(* PLC project Generated.project, CODESYS CODESYS V3.5 SP19 Patch 1 *)
(* stored: creationDateTime 2026-09-06T13:00:42.431888, modificationDateTime 2026-09-06T13:00:42.431888 *)

(* ======================================================================= ⚖️ ST_fbWinch_Symmetry_Cfg — Configuration des seuils de symétrie M1/M2 ─────────────────────────────────────────────────────────────── 🎯 Rôle : Seuils de tolérance pour le diagnostic passif de symétrie treuils 📄 Doc métier : DOC/AF/AF_Partie-10_Fonction_Winch_v2.1.md ======================================================================= *)
TYPE ST_fbWinch_Symmetry_Cfg : STRUCT
  DeltaStartDelay_Ms : UDINT := 100;  (* Ecart max tolere au demarrage (ms) *)
  DeltaBrakeReleaseTime_Ms : UDINT := 100;  (* Ecart max temps desserrage frein (ms) *)
  DeltaBrakeApplyTime_Ms : UDINT := 100;  (* Ecart max temps serrage frein (ms) *)
  DeltaStopDistance_Mm : UDINT := 100;  (* Ecart max distance d'arret (mm) *)
  DeltaStopTime_Ms : UDINT := 200;  (* Ecart max temps d'arret (ms) *)
  MinimumCommandTime_Ms : UDINT := 1000;  (* Duree minimale de commande pour qualification (ms) *)
  MinimumSpeed_Mps : REAL := 0.05;  (* Vitesse minimale pour qualification (m/s) *)
END_STRUCT;
END_TYPE

(* ======================================================================= 📊 ST_fbWinch_Symmetry_Data — Données mesurées de symétrie M1/M2 ─────────────────────────────────────────────────────────────── 🎯 Rôle : Structure des résultats de mesures et d'écarts du diagnostic symétrie 📄 Doc métier : DOC/AF/AF_Partie-10_Fonction_Winch_v2.1.md ======================================================================= *)
TYPE ST_fbWinch_Symmetry_Data : STRUCT
  DeltaStartDelay_Ms : UDINT;  (* Ecart mesure au demarrage (ms) *)
  DeltaBrakeReleaseTime_Ms : UDINT;  (* Ecart mesure temps desserrage frein (ms) *)
  DeltaBrakeApplyTime_Ms : UDINT;  (* Ecart mesure temps serrage frein (ms) *)
  DeltaStopDistance_Mm : UDINT;  (* Ecart mesure distance d'arret (mm) *)
  DeltaStopTime_Ms : UDINT;  (* Ecart mesure temps d'arret (ms) *)
  MaxSyncDeviation_M : REAL;  (* Ecart maximal de synchronisme enregistre (m) *)
END_STRUCT;
END_TYPE

(* ======================================================================= ⚖️ FB_Winch_Symmetry — Mesure passive M1/M2 ─────────────────────────────────────────────────────────────── 🎯 Rôle : Observateur de symétrie et de synchronisme des treuils M1/M2 📄 Doc métier : DOC/AF/AF_Partie-10_Fonction_Winch_v2.1.md 🔒 Observateur pur : Aucune ecriture de commande, securite ou mouvement ======================================================================= *)
FUNCTION_BLOCK FB_Winch_Symmetry
  VAR_INPUT
    Reset : BOOL;  (* === COMMANDES ET CONSIGNES === --> [CMD] Reinitialisation des mesures sur front *)
    M1CommandActive : BOOL;  (* --> [CMD] Commande active sur treuil M1 *)
    M2CommandActive : BOOL;  (* --> [CMD] Commande active sur treuil M2 *)
    M1Direction : INT;  (* --> [CMD] Sens commande M1 (-1/0/+1) *)
    M2Direction : INT;  (* --> [CMD] Sens commande M2 (-1/0/+1) *)
    M1BrakeCmd : BOOL;  (* === FEEDBACKS HARWARE ET FREINS === --> [HW] Ordre ouverture frein M1 *)
    M2BrakeCmd : BOOL;  (* --> [HW] Ordre ouverture frein M2 *)
    M1BrakeApplied : BOOL;  (* --> [HW] Etat frein M1 serre *)
    M2BrakeApplied : BOOL;  (* --> [HW] Etat frein M2 serre *)
    M1Position_M : REAL;  (* === MESURES POSITIONS ET VITESSES === --> [HW] Position mesuree M1 (m) *)
    M2Position_M : REAL;  (* --> [HW] Position mesuree M2 (m) *)
    M1Speed_Mps : REAL;  (* --> [HW] Vitesse mesuree M1 (m/s) *)
    M2Speed_Mps : REAL;  (* --> [HW] Vitesse mesuree M2 (m/s) *)
    SyncDeviation_M : REAL;  (* --> [HW] Ecart instantane synchro (m) *)
    Config : ST_fbWinch_Symmetry_Cfg;  (* === CONFIGURATION === --> [CFG] Configuration des seuils de symetrie *)
  END_VAR
  VAR_OUTPUT
    SymmetryOk : BOOL;  (* === ETATS IEC ET SYNOPTIQUE === <-- [STAT] Symetrie globale conforme aux criteres *)
    SymmetryValid : BOOL;  (* <-- [STAT] Mesure de symetrie valide et calculee *)
  END_VAR
  VAR_IN_OUT
    Data : ST_fbWinch_Symmetry_Data;  (* === STRUCTURES DE DONNÉES PARTAGÉES === <-> [BUS] Donnees de mesures de symetrie *)
  END_VAR
  VAR
    ResetEdge : R_TRIG;  (* === SOUS-INSTANCES FB === * [INST] Detecteur front reinitialisation *)
    CycleTime : FB_CycleTime;  (* * [INST] Calcul du temps de cycle *)
    CommandTon : TON;  (* === TIMERS INTERNES === . [LOC] Tempo qualification commande stable *)
    MotionTimer : TON;  (* . [LOC] Chronometre de mouvement *)
    StopTimer : TON;  (* . [LOC] Chronometre d'arret *)
    Comparable : BOOL;  (* === VARIABLES LOCALES CALCULÉES === . [LOC] Conditions de comparaison remplies *)
    Qualified : BOOL;  (* . [LOC] Phase de mesure qualifiee *)
    PreviousQualified : BOOL;  (* . [LOC] Etat qualifie cycle precedent *)
    Stopping : BOOL;  (* . [LOC] Phase d'arret en cours *)
    StartCapturedM1 : BOOL;  (* . [LOC] Top depart capture M1 *)
    StartCapturedM2 : BOOL;  (* . [LOC] Top depart capture M2 *)
    StopCapturedM1 : BOOL;  (* . [LOC] Top arret capture M1 *)
    StopCapturedM2 : BOOL;  (* . [LOC] Top arret capture M2 *)
    StartMsM1 : UDINT;  (* . [LOC] Horodatage d'ouverture M1 (ms) *)
    StartMsM2 : UDINT;  (* . [LOC] Horodatage d'ouverture M2 (ms) *)
    ReleaseMsM1 : UDINT;  (* . [LOC] Temps de desserrage frein M1 (ms) *)
    ReleaseMsM2 : UDINT;  (* . [LOC] Temps de desserrage frein M2 (ms) *)
    ApplyMsM1 : UDINT;  (* . [LOC] Temps de serrage frein M1 (ms) *)
    ApplyMsM2 : UDINT;  (* . [LOC] Temps de serrage frein M2 (ms) *)
    StopMsM1 : UDINT;  (* . [LOC] Horodatage d'arret M1 (ms) *)
    StopMsM2 : UDINT;  (* . [LOC] Horodatage d'arret M2 (ms) *)
    StopStartM1_M : REAL;  (* . [LOC] Position debut d'arret M1 (m) *)
    StopStartM2_M : REAL;  (* . [LOC] Position debut d'arret M2 (m) *)
  END_VAR

            

{region "§1 Reset et qualification"}
CycleTime(DefaultValueS := 0.010); ResetEdge(CLK := Reset);
IF ResetEdge.Q THEN Data.DeltaStartDelay_Ms:=0; Data.DeltaBrakeReleaseTime_Ms:=0; Data.DeltaBrakeApplyTime_Ms:=0; Data.DeltaStopDistance_Mm:=0; Data.DeltaStopTime_Ms:=0; Data.MaxSyncDeviation_M:=0.0; END_IF;
Comparable := M1CommandActive AND M2CommandActive AND (M1Direction = M2Direction) AND (M1Direction <> 0);
CommandTon(IN := Comparable, PT := UDINT_TO_TIME(Config.MinimumCommandTime_Ms));
Qualified := CommandTon.Q AND (M1Speed_Mps >= Config.MinimumSpeed_Mps) AND (M2Speed_Mps >= Config.MinimumSpeed_Mps);
MotionTimer(IN := Comparable, PT := T#1h);
StopTimer(IN := Stopping, PT := T#1h);
IF NOT Comparable THEN StartCapturedM1:=FALSE; StartCapturedM2:=FALSE; ReleaseMsM1:=0; ReleaseMsM2:=0; ApplyMsM1:=0; ApplyMsM2:=0; END_IF;
IF Comparable AND (M1Speed_Mps >= Config.MinimumSpeed_Mps) AND NOT StartCapturedM1 THEN StartMsM1:=TIME_TO_UDINT(MotionTimer.ET); StartCapturedM1:=TRUE; END_IF;
IF Comparable AND (M2Speed_Mps >= Config.MinimumSpeed_Mps) AND NOT StartCapturedM2 THEN StartMsM2:=TIME_TO_UDINT(MotionTimer.ET); StartCapturedM2:=TRUE; END_IF;
{endregion}

{region "§2 Mesure symétrie"}
IF Qualified THEN
    IF M1BrakeCmd AND M1BrakeApplied THEN ReleaseMsM1 := ReleaseMsM1 + REAL_TO_UDINT(CycleTime.CycleTimeS * 1000.0); END_IF;
    IF M2BrakeCmd AND M2BrakeApplied THEN ReleaseMsM2 := ReleaseMsM2 + REAL_TO_UDINT(CycleTime.CycleTimeS * 1000.0); END_IF;
    IF NOT M1BrakeCmd AND NOT M1BrakeApplied THEN ApplyMsM1 := ApplyMsM1 + REAL_TO_UDINT(CycleTime.CycleTimeS * 1000.0); END_IF;
    IF NOT M2BrakeCmd AND NOT M2BrakeApplied THEN ApplyMsM2 := ApplyMsM2 + REAL_TO_UDINT(CycleTime.CycleTimeS * 1000.0); END_IF;
    IF SyncDeviation_M > Data.MaxSyncDeviation_M THEN Data.MaxSyncDeviation_M := SyncDeviation_M; END_IF;
END_IF;
IF PreviousQualified AND NOT Comparable THEN Stopping:=TRUE; StopCapturedM1:=FALSE; StopCapturedM2:=FALSE; StopStartM1_M:=M1Position_M; StopStartM2_M:=M2Position_M; END_IF;
IF Stopping THEN
    IF (M1Speed_Mps < Config.MinimumSpeed_Mps) AND NOT StopCapturedM1 THEN StopMsM1:=TIME_TO_UDINT(StopTimer.ET); StopCapturedM1:=TRUE; END_IF;
    IF (M2Speed_Mps < Config.MinimumSpeed_Mps) AND NOT StopCapturedM2 THEN StopMsM2:=TIME_TO_UDINT(StopTimer.ET); StopCapturedM2:=TRUE; END_IF;
    IF StopCapturedM1 AND StopCapturedM2 THEN
        Data.DeltaStartDelay_Ms := DINT_TO_UDINT(ABS(UDINT_TO_DINT(StartMsM1) - UDINT_TO_DINT(StartMsM2)));
        Data.DeltaBrakeReleaseTime_Ms := DINT_TO_UDINT(ABS(UDINT_TO_DINT(ReleaseMsM1) - UDINT_TO_DINT(ReleaseMsM2)));
        Data.DeltaBrakeApplyTime_Ms := DINT_TO_UDINT(ABS(UDINT_TO_DINT(ApplyMsM1) - UDINT_TO_DINT(ApplyMsM2)));
        Data.DeltaStopDistance_Mm := REAL_TO_UDINT(ABS(ABS(M1Position_M - StopStartM1_M) - ABS(M2Position_M - StopStartM2_M)) * 1000.0);
        Data.DeltaStopTime_Ms := DINT_TO_UDINT(ABS(UDINT_TO_DINT(StopMsM1) - UDINT_TO_DINT(StopMsM2))); Stopping := FALSE; SymmetryValid := TRUE;
    END_IF;
END_IF;
{endregion}

{region "§3 Sortie"}
SymmetryOk := SymmetryValid AND (Data.DeltaStartDelay_Ms<=Config.DeltaStartDelay_Ms) AND (Data.DeltaBrakeReleaseTime_Ms<=Config.DeltaBrakeReleaseTime_Ms) AND (Data.DeltaBrakeApplyTime_Ms<=Config.DeltaBrakeApplyTime_Ms) AND (Data.DeltaStopDistance_Mm<=Config.DeltaStopDistance_Mm) AND (Data.DeltaStopTime_Ms<=Config.DeltaStopTime_Ms);
PreviousQualified := Qualified;
{endregion}

          
END_FUNCTION_BLOCK

(* ======================================================================= ⚙️ FB_CycleTime — Mesure du temps de cycle réel de la tâche ─────────────────────────────────────────────────────────────── 🎯 Rôle : Calcul du dt réel entre deux exécutions successives ⚙️ Calcul : Delta horloge système TIME() converti en secondes 🛡️ Robustesse : dt borné (0 < dt <= CST_MaxCycleDeltaMs) sinon valeur de secours — neutralise les artefacts de rebouclage TIME() (49,7 j) et de reprise (online-change, debug) 📄 Doc métier : DOC/AF/AF_Partie-03_Contrats_Composants/FB_CycleTime_v1.0.md ======================================================================= *)
FUNCTION_BLOCK FB_CycleTime
  VAR_INPUT
    DefaultValueS : REAL := 0.004;  (* === REGLAGES DE SECOURS === --> [CFG] Valeur de secours par defaut (ex: 4ms = 0.004s) *)
  END_VAR
  VAR_OUTPUT
    CycleTimeS : REAL;  (* === MESURE ET DIAGNOSTIC === <-- [DIAG] Temps ecoule reel calcule (secondes) *)
  END_VAR
  VAR
    TimeCurrent : TIME;  (* === HORLOGE ET MEMOIRE TEMPORELLE === . [LOC] Temps systeme actuel *)
    TimeLast : TIME;  (* . [LOC] Empreinte de temps du cycle precedent *)
    DeltaTimeMs : UDINT;  (* . [LOC] Ecart brut calcule (ms) *)
    InitDone : BOOL;  (* . [LOC] Drapeau d'initialisation du premier cycle *)
    CST_MaxCycleDeltaMs : UDINT := 1000;  (* === BORNE HAUTE DU DELTA DE CYCLE === Plafond physique du dt entre deux scans (ms) : au-dela -> valeur de secours *)
  END_VAR

            

{region "§1 Acquisition temps"}
// 1. ACQUISITION DU TEMPS SYSTÈME
TimeCurrent := TIME();
{endregion}

{region "§2 Initialisation"}
// 2. INITIALISATION UNIQUE AU PREMIER CYCLE
IF NOT InitDone THEN
    TimeLast := TimeCurrent;
    InitDone := TRUE;
    CycleTimeS := DefaultValueS;
    RETURN;
END_IF;
{endregion}

{region "§3 Calcul delta"}
// 3. CALCUL DU DELTA EN MILLISECONDES
DeltaTimeMs := TIME_TO_UDINT(TimeCurrent - TimeLast);
{endregion}

{region "§4 Conversion, secours et bornage"}
// 4. CONVERSION EN SECONDES, AVEC DOUBLE BORNAGE DU DELTA
//
// TIME() est un compteur systeme 32 bits en millisecondes depuis le demarrage de
// l'automate. Il n'est PAS absolu : il reboucle a 0 tous les 2^32 ms (~49,7 jours).
// La soustraction TimeCurrent - TimeLast est modulo 2^32 : au passage du rebouclage,
// tant que l'ecart reel entre deux scans reste < 49,7 j (toujours vrai a 10 ms),
// DeltaTimeMs reste correct. Le rebouclage seul n'est donc pas le risque principal.
//
// Le vrai risque est un DeltaTimeMs REELLEMENT > CST_MaxCycleDeltaMs : reprise apres
// un online-change, sortie d'un point d'arret / pas-a-pas debug, ou fenetre du
// rebouclage TIME(). Le chien de garde tache (200 ms, sensibilite 1) borne deja les
// gels en fonctionnement ; ce plafond couvre les cas hors surveillance.
// Un dt aberrant publie tel quel donnerait un CycleTimeS enorme, propage en un seul
// scan dans les rampes de vitesse et les integrateurs de position/frein -> saut
// physique. Fail-safe : hors de la plage nominale (0 < dt <= plafond), on publie la
// valeur de secours DefaultValueS au lieu de l'artefact. Pas de redemarrage auto.
//
// Borne basse dt = 0 (anti-zero, ex. premier appel du scan) et borne haute
// dt > CST_MaxCycleDeltaMs (anti-artefact) partagent la meme branche de secours.
IF (DeltaTimeMs > 0) AND (DeltaTimeMs <= CST_MaxCycleDeltaMs) THEN
    CycleTimeS := UDINT_TO_REAL(DeltaTimeMs) / 1000.0;
ELSE
    CycleTimeS := DefaultValueS;
END_IF;
{endregion}

{region "§5 Archivage"}
// 5. ARCHIVAGE POUR LE PROCHAIN CYCLE
TimeLast := TimeCurrent;
{endregion}

          
END_FUNCTION_BLOCK
